TYPE T_Ctrl_SIf_ICL_In :
STRUCT
	Module: T_Ctrl_SIf_MOD_In;
END_STRUCT
END_TYPE

(* stored: Version 1.1.0.1, ProductVersion 3.1.0.19
   DUT T_Ctrl_SIf_ICL_In: Id {99517368-6fda-497b-a561-18a29e36ceea} *)
